INTERFACE I_DatatypeAddedEvent EXTENDS I_Event

PROPERTY PUBLIC Target : I_Datatype
GET
END_GET
END_PROPERTY

END_INTERFACE

(* stored: Version 1.1.0.1, ProductVersion 3.1.4024.12
   Itf I_DatatypeAddedEvent: Id {3d317bc9-7c43-429f-b510-7d219205f094}
   Property Target: Id {ba87f871-f05f-4cd2-9b14-83a0008376f8}
   Get Get: Id {de678589-f467-4ab2-a9ae-409e01e30506} *)
